/// Implicitly generated code : DO NOT EDIT!!!
/// Checks for division by 0, if divisor is 0, replace it with 1 and report error
{attribute 'no_check' := ''}
{attribute 'check_div_real64' := ''}
FUNCTION CheckDivLReal : LREAL
VAR_INPUT
	divisor: LREAL;
END_VAR

IF divisor = 0 THEN
	// replace divisor and report error if necessary
	CheckDivLReal := 1;
	GVL_Supervision.aCodeErr[eCodeError_divLReal] := TRUE;
ELSE
	CheckDivLReal:=divisor;
END_IF;

END_FUNCTION

(* stored: Version 1.1.0.1, ProductVersion 3.1.4022.9
   POU CheckDivLReal: Id {edede5d0-b496-4d01-bb77-d66fb2dbae07}, SpecialFunc None *)
